(* CoDeSys 2.3 export: PLC_PRG.EXP *)

(* POU PLC_PRG, LD *)
PROGRAM PLC_PRG
VAR
	S0 AT %MX1.0: BOOL;
	CH AT %IX0.1: BOOL;
	SP AT %IX0.0: BOOL;
	QCU AT %MX0.1: BOOL;
	T0 AT %MX2.0: BOOL;
	S1 AT %MX1.1: BOOL;
	T1 AT %MX2.1: BOOL;
	S2 AT %MX1.2: BOOL;
	T2 AT %MX2.2: BOOL;
	S3 AT %MX1.3: BOOL;
	QT1 AT %MX0.3: BOOL;
	T3 AT %MX2.3: BOOL;
	S4 AT %MX1.4: BOOL;
	T4 AT %MX2.4: BOOL;
	CA AT %QX0.0: BOOL;
	CB AT %QX0.1: BOOL;
	CC AT %QX0.2: BOOL;
	M AT %QX0.3: BOOL;
	CU AT %MX0.0: BOOL;
	P: R_TRIG;
	T1_EN AT %MX0.2: BOOL;
	TEMPORIZADOR1: TON;
	CTU: CTU;
	COUNT AT %MW10: INT;
END_VAR
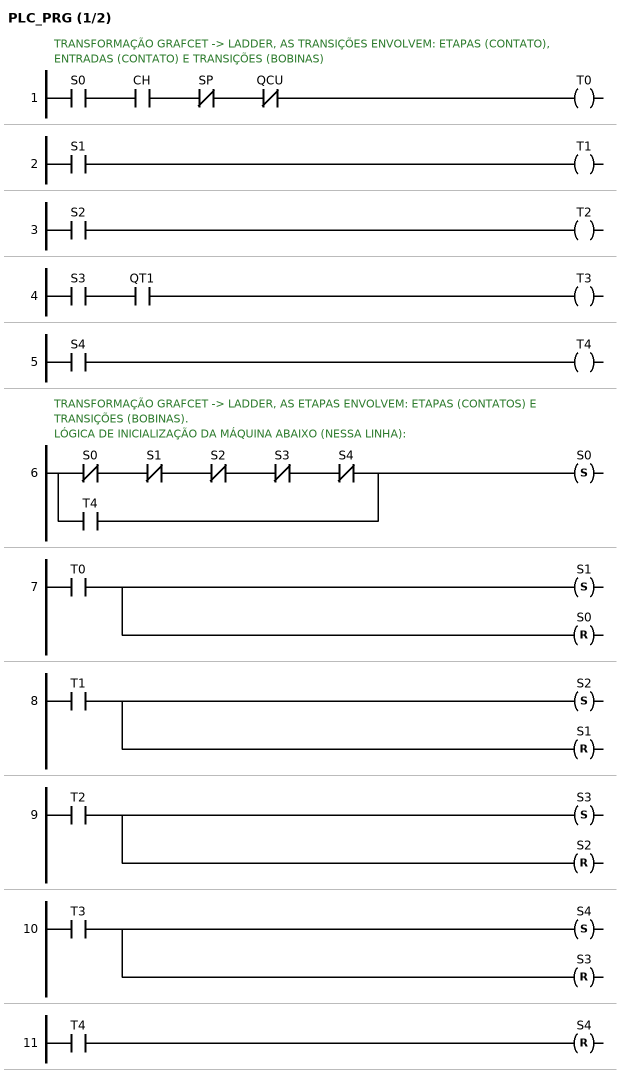
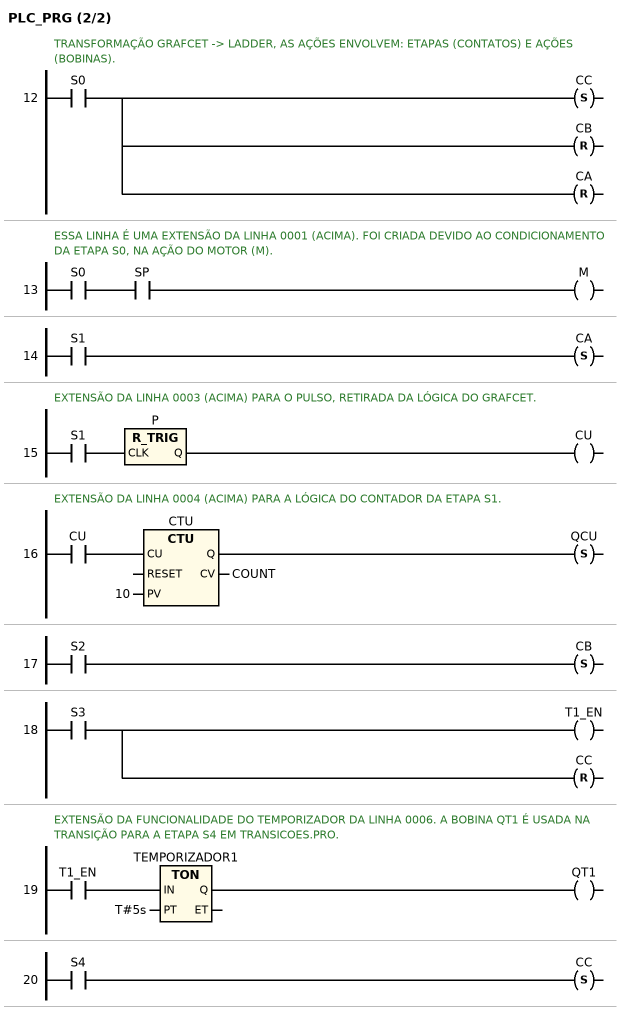
_LD_ (* Ladder Diagram *)
NETWORK 1 (* TRANSFORMAÇÃO GRAFCET -> LADDER, AS TRANSIÇÕES ENVOLVEM: ETAPAS (CONTATO), ENTRADAS (CONTATO) E TRANSIÇÕES (BOBINAS) *)
	[S0] - [CH] - [/SP] - [/QCU] --- (T0)
NETWORK 2
	[S1] --- (T1)
NETWORK 3
	[S2] --- (T2)
NETWORK 4
	[S3] - [QT1] --- (T3)
NETWORK 5
	[S4] --- (T4)
NETWORK 6 (* TRANSFORMAÇÃO GRAFCET -> LADDER, AS ETAPAS ENVOLVEM: ETAPAS (CONTATOS) E TRANSIÇÕES (BOBINAS). / LÓGICA DE INICIALIZAÇÃO DA MÁQUINA ABAIXO (NESSA LINHA): *)
	{ [/S0] - [/S1] - [/S2] - [/S3] - [/S4] | [T4] } --- (S S0)
NETWORK 7
	[T0] --- (S S1) (R S0)
NETWORK 8
	[T1] --- (S S2) (R S1)
NETWORK 9
	[T2] --- (S S3) (R S2)
NETWORK 10
	[T3] --- (S S4) (R S3)
NETWORK 11
	[T4] --- (R S4)
NETWORK 12 (* TRANSFORMAÇÃO GRAFCET -> LADDER, AS AÇÕES ENVOLVEM: ETAPAS (CONTATOS) E AÇÕES (BOBINAS). *)
	[S0] --- (S CC) (R CB) (R CA)
NETWORK 13 (* ESSA LINHA É UMA EXTENSÃO DA LINHA 0001 (ACIMA). FOI CRIADA DEVIDO AO CONDICIONAMENTO DA ETAPA S0, NA AÇÃO DO MOTOR (M). *)
	[S0] - [SP] --- (M)
NETWORK 14
	[S1] --- (S CA)
NETWORK 15 (* EXTENSÃO DA LINHA 0003 (ACIMA) PARA O PULSO, RETIRADA DA LÓGICA DO GRAFCET. *)
	[S1] - P:R_TRIG(CLK: *) --- (CU)
NETWORK 16 (* EXTENSÃO DA LINHA 0004 (ACIMA) PARA A LÓGICA DO CONTADOR DA ETAPA S1. *)
	[CU] - CTU:CTU(CU: *, RESET: , PV: 10, CV => COUNT) --- (S QCU)
NETWORK 17
	[S2] --- (S CB)
NETWORK 18
	[S3] --- (T1_EN) (R CC)
NETWORK 19 (* EXTENSÃO DA FUNCIONALIDADE DO TEMPORIZADOR DA LINHA 0006. A BOBINA QT1 É USADA NA TRANSIÇÃO PARA A ETAPA S4 EM TRANSICOES.PRO. *)
	[T1_EN] - TEMPORIZADOR1:TON(IN: *, PT: T#5s) --- (QT1)
NETWORK 20
	[S4] --- (S CC)
_END_LD_
(* the same logic as Structured Text *)
(* Network 1 *)
T0 := S0 AND CH AND NOT SP AND NOT QCU;
(* Network 2 *)
T1 := S1;
(* Network 3 *)
T2 := S2;
(* Network 4 *)
T3 := S3 AND QT1;
(* Network 5 *)
T4 := S4;
(* Network 6 *)
IF NOT S0 AND NOT S1 AND NOT S2 AND NOT S3 AND NOT S4 OR T4 THEN S0 := TRUE; END_IF;
(* Network 7 *)
IF T0 THEN S1 := TRUE; S0 := FALSE; END_IF;
(* Network 8 *)
IF T1 THEN S2 := TRUE; S1 := FALSE; END_IF;
(* Network 9 *)
IF T2 THEN S3 := TRUE; S2 := FALSE; END_IF;
(* Network 10 *)
IF T3 THEN S4 := TRUE; S3 := FALSE; END_IF;
(* Network 11 *)
IF T4 THEN S4 := FALSE; END_IF;
(* Network 12 *)
IF S0 THEN CC := TRUE; CB := FALSE; CA := FALSE; END_IF;
(* Network 13 *)
M := S0 AND SP;
(* Network 14 *)
IF S1 THEN CA := TRUE; END_IF;
(* Network 15 *)
P(CLK := S1);
CU := P.Q;
(* Network 16: see the listing above *)
(* Network 17 *)
IF S2 THEN CB := TRUE; END_IF;
(* Network 18 *)
T1_EN := S3;
IF S3 THEN CC := FALSE; END_IF;
(* Network 19 *)
TEMPORIZADOR1(IN := T1_EN, PT := T#5s);
QT1 := TEMPORIZADOR1.Q;
(* Network 20 *)
IF S4 THEN CC := TRUE; END_IF;
END_PROGRAM
ACTION ACOES:
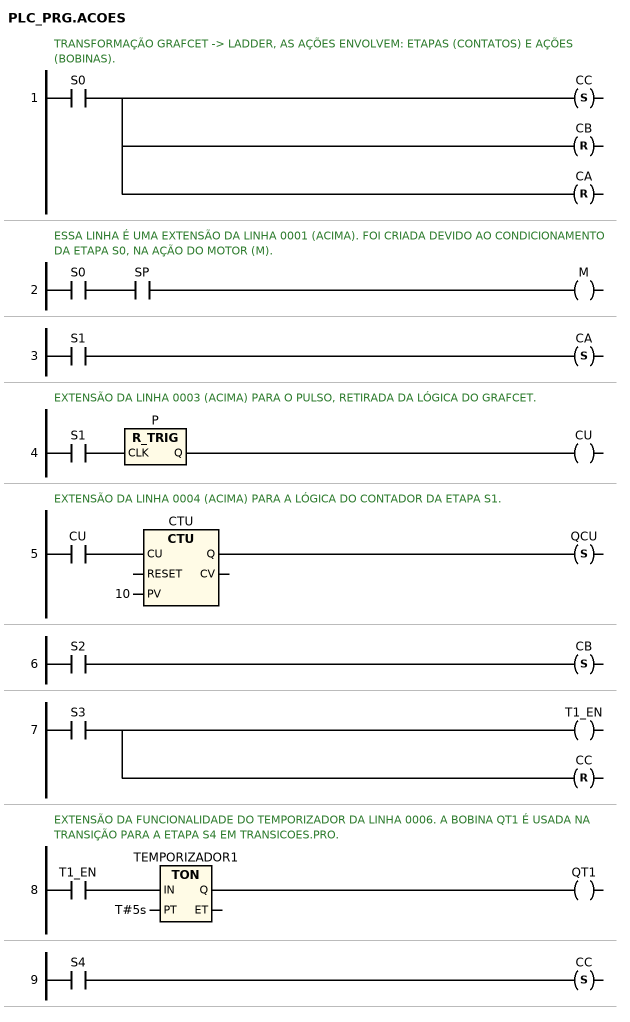
_LD_ (* Ladder Diagram *)
NETWORK 1 (* TRANSFORMAÇÃO GRAFCET -> LADDER, AS AÇÕES ENVOLVEM: ETAPAS (CONTATOS) E AÇÕES (BOBINAS). *)
	[S0] --- (S CC) (R CB) (R CA)
NETWORK 2 (* ESSA LINHA É UMA EXTENSÃO DA LINHA 0001 (ACIMA). FOI CRIADA DEVIDO AO CONDICIONAMENTO DA ETAPA S0, NA AÇÃO DO MOTOR (M). *)
	[S0] - [SP] --- (M)
NETWORK 3
	[S1] --- (S CA)
NETWORK 4 (* EXTENSÃO DA LINHA 0003 (ACIMA) PARA O PULSO, RETIRADA DA LÓGICA DO GRAFCET. *)
	[S1] - P:R_TRIG(CLK: *) --- (CU)
NETWORK 5 (* EXTENSÃO DA LINHA 0004 (ACIMA) PARA A LÓGICA DO CONTADOR DA ETAPA S1. *)
	[CU] - CTU:CTU(CU: *, RESET: , PV: 10) --- (S QCU)
NETWORK 6
	[S2] --- (S CB)
NETWORK 7
	[S3] --- (T1_EN) (R CC)
NETWORK 8 (* EXTENSÃO DA FUNCIONALIDADE DO TEMPORIZADOR DA LINHA 0006. A BOBINA QT1 É USADA NA TRANSIÇÃO PARA A ETAPA S4 EM TRANSICOES.PRO. *)
	[T1_EN] - TEMPORIZADOR1:TON(IN: *, PT: T#5s) --- (QT1)
NETWORK 9
	[S4] --- (S CC)
_END_LD_
(* the same logic as Structured Text *)
(* Network 1 *)
IF S0 THEN CC := TRUE; CB := FALSE; CA := FALSE; END_IF;
(* Network 2 *)
M := S0 AND SP;
(* Network 3 *)
IF S1 THEN CA := TRUE; END_IF;
(* Network 4 *)
P(CLK := S1);
CU := P.Q;
(* Network 5: see the listing above *)
(* Network 6 *)
IF S2 THEN CB := TRUE; END_IF;
(* Network 7 *)
T1_EN := S3;
IF S3 THEN CC := FALSE; END_IF;
(* Network 8 *)
TEMPORIZADOR1(IN := T1_EN, PT := T#5s);
QT1 := TEMPORIZADOR1.Q;
(* Network 9 *)
IF S4 THEN CC := TRUE; END_IF;
END_ACTION
ACTION ETAPAS:
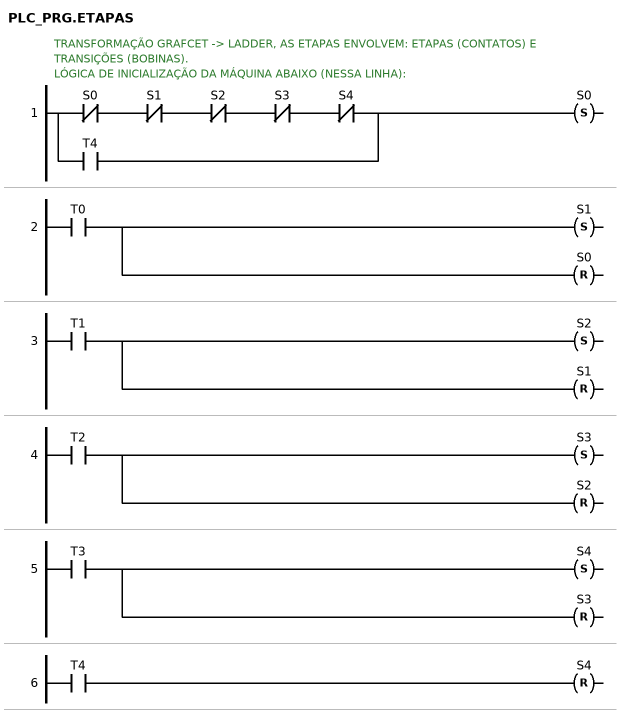
_LD_ (* Ladder Diagram *)
NETWORK 1 (* TRANSFORMAÇÃO GRAFCET -> LADDER, AS ETAPAS ENVOLVEM: ETAPAS (CONTATOS) E TRANSIÇÕES (BOBINAS). / LÓGICA DE INICIALIZAÇÃO DA MÁQUINA ABAIXO (NESSA LINHA): *)
	{ [/S0] - [/S1] - [/S2] - [/S3] - [/S4] | [T4] } --- (S S0)
NETWORK 2
	[T0] --- (S S1) (R S0)
NETWORK 3
	[T1] --- (S S2) (R S1)
NETWORK 4
	[T2] --- (S S3) (R S2)
NETWORK 5
	[T3] --- (S S4) (R S3)
NETWORK 6
	[T4] --- (R S4)
_END_LD_
(* the same logic as Structured Text *)
(* Network 1: TRANSFORMAÇÃO GRAFCET -> LADDER, AS ETAPAS ENVOLVEM: ETAPAS (CONTATOS) E TRANSIÇÕES (BOBINAS). / LÓGICA DE INICIALIZAÇÃO DA MÁQUINA ABAIXO (NESSA LINHA): *)
IF NOT S0 AND NOT S1 AND NOT S2 AND NOT S3 AND NOT S4 OR T4 THEN S0 := TRUE; END_IF;
(* Network 2 *)
IF T0 THEN S1 := TRUE; S0 := FALSE; END_IF;
(* Network 3 *)
IF T1 THEN S2 := TRUE; S1 := FALSE; END_IF;
(* Network 4 *)
IF T2 THEN S3 := TRUE; S2 := FALSE; END_IF;
(* Network 5 *)
IF T3 THEN S4 := TRUE; S3 := FALSE; END_IF;
(* Network 6 *)
IF T4 THEN S4 := FALSE; END_IF;
END_ACTION
ACTION TRANSICOES:
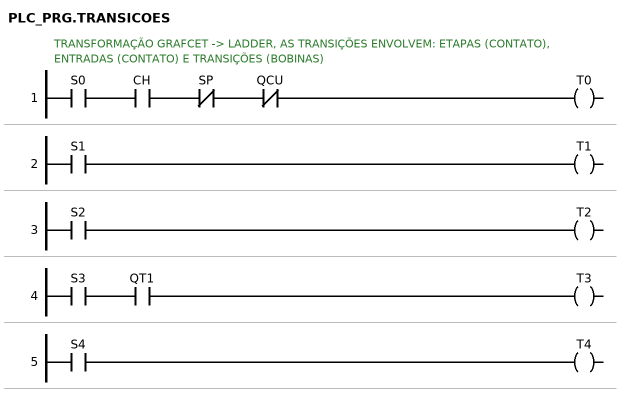
_LD_ (* Ladder Diagram *)
NETWORK 1 (* TRANSFORMAÇÃO GRAFCET -> LADDER, AS TRANSIÇÕES ENVOLVEM: ETAPAS (CONTATO), ENTRADAS (CONTATO) E TRANSIÇÕES (BOBINAS) *)
	[S0] - [CH] - [/SP] - [/QCU] --- (T0)
NETWORK 2
	[S1] --- (T1)
NETWORK 3
	[S2] --- (T2)
NETWORK 4
	[S3] - [QT1] --- (T3)
NETWORK 5
	[S4] --- (T4)
_END_LD_
(* the same logic as Structured Text *)
(* Network 1: TRANSFORMAÇÃO GRAFCET -> LADDER, AS TRANSIÇÕES ENVOLVEM: ETAPAS (CONTATO), ENTRADAS (CONTATO) E TRANSIÇÕES (BOBINAS) *)
T0 := S0 AND CH AND NOT SP AND NOT QCU;
(* Network 2 *)
T1 := S1;
(* Network 3 *)
T2 := S2;
(* Network 4 *)
T3 := S3 AND QT1;
(* Network 5 *)
T4 := S4;
END_ACTION
